VAR_GLOBAL
	//Better have your inputs and outputs!
	Serial_P1_stComIn   AT %I*	:	EL6inData22B (*KL6inData22B*);
	Serial_P1_stComOut  AT %Q*	:	EL6outData22B (*KL6outData22B*);
	Serial_P1_SerialTXBuffer :ComBuffer;
	Serial_P1_SerialRXBuffer :ComBuffer;
	
END_VAR

(* stored: Version 1.1.0.1, ProductVersion 3.1.4020.12
   GVL GVL_SerialIO: Id {e2338c89-1965-407c-b604-590f80e0dc24} *)
